SUBAPPLICATION Uebung_019a (* Umschalten einer Maske *)
  (* Standard: 61499-2; Description: Copyright (c) 2023 Meisterschulen am Ostbahnhof This program and the accompanying materials are made available under the terms of the Eclipse Public License 2.0 which is available at https://www.eclipse.org/legal/epl-2.0/ SPDX-License-Identifier: EPL-2.0 *)
  (* Version 1.0, 2023-10-23, Franz Höpfinger, Meisterschulen am Ostbahnhof *)
  PACKAGE Uebungen;
  IMPORT SoftKeyActivationCode::SK_PRESSED;
  IMPORT Uebungen::const::UT::DefaultPool::AlarmMask_A2_medium;
  IMPORT Uebungen::const::UT::DefaultPool::DataMask_M1;
  IMPORT Uebungen::const::UT::DefaultPool::DataMask_M2;
  IMPORT Uebungen::const::UT::DefaultPool::WorkingSet_0;
  IMPORT isobus::ut::IDs::ID_NULL;
  IMPORT logiBUS::io::DI::logiBUS_DI::Input_I1;
  IMPORT logiBUS::io::DI::logiBUS_DI::Input_I2;
  IMPORT logiBUS::io::DI::logiBUS_DI::Input_I3;
  IMPORT logiBUS::io::DI::logiBUS_DI_Events::BUTTON_SINGLE_CLICK;
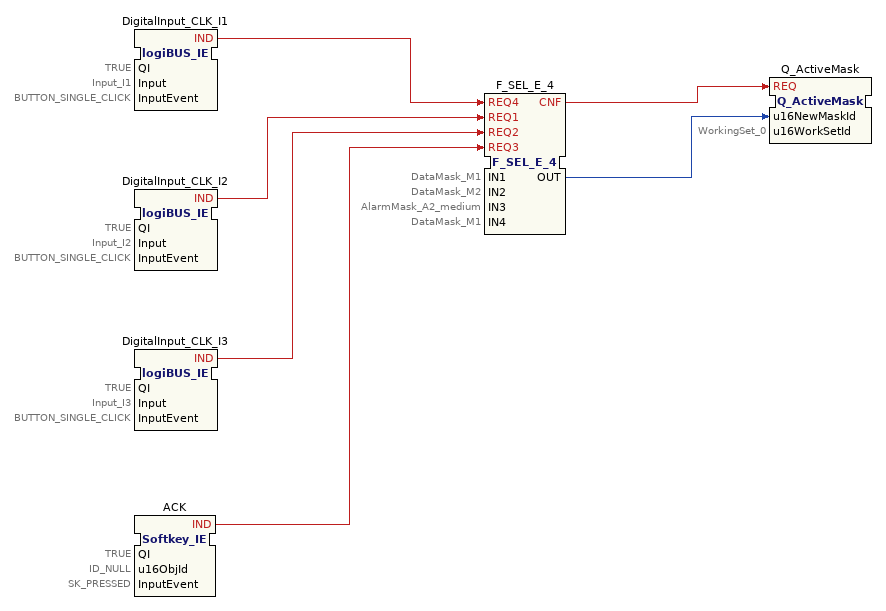
  FBS
    DigitalInput_CLK_I1 : logiBUS::io::DI::logiBUS_IE(QI := TRUE, Input := Input_I1, InputEvent := BUTTON_SINGLE_CLICK);
    Q_ActiveMask : isobus::ut::Q_ActiveMask(u16WorkSetId := WorkingSet_0);
    DigitalInput_CLK_I2 : logiBUS::io::DI::logiBUS_IE(QI := TRUE, Input := Input_I2, InputEvent := BUTTON_SINGLE_CLICK);
    F_SEL_E_4 : eclipse4diac::utils::selection::F_SEL_E_4(IN1 := DataMask_M1, IN2 := DataMask_M2, IN3 := AlarmMask_A2_medium, IN4 := DataMask_M1);
    DigitalInput_CLK_I3 : logiBUS::io::DI::logiBUS_IE(QI := TRUE, Input := Input_I3, InputEvent := BUTTON_SINGLE_CLICK);
    ACK : Softkey_IE(QI := TRUE, u16ObjId := ID_NULL, InputEvent := SK_PRESSED);
  END_FBS
  EVENT_CONNECTIONS
    DigitalInput_CLK_I1.IND TO F_SEL_E_4.REQ4;
    DigitalInput_CLK_I2.IND TO F_SEL_E_4.REQ1;
    F_SEL_E_4.CNF TO Q_ActiveMask.REQ;
    DigitalInput_CLK_I3.IND TO F_SEL_E_4.REQ2;
    ACK.IND TO F_SEL_E_4.REQ3;
  END_CONNECTIONS
  DATA_CONNECTIONS
    F_SEL_E_4.OUT TO Q_ActiveMask.u16NewMaskId;
  END_CONNECTIONS
END_SUBAPPLICATION
